TYPE teCTCWarningID :
(
	CTC_WARNING_OK 				:= 0,
	CTC_WARNING_FB_SETPOINTS 	:= 1,
	CTC_WARNING_FB_COMMAND 		:= 2,
	CTC_WARNING_EVENT 			:= 3
);
END_TYPE

(* stored: Version 1.1.0.1, ProductVersion 3.1.4026.17
   EnumerationTextList teCTCWarningID: Id {da05a0eb-7045-42f5-b279-45cefdf19dc8} *)
